TYPE ST_TCUEPT :
STRUCT
	// LoadPort module state 
	//arrLPSubModule : ARRAY [1..(.NO_OF_LANES)] OF ST_LP_SubModuleEPT;
	// Vision Shuttle 
	TCU : E_EPT;
END_STRUCT
END_TYPE

(* stored: Version 1.1.0.1, ProductVersion 3.1.4022.12
   DUT ST_TCUEPT: Id {9f00026a-a904-41aa-bc64-905de90e5a87} *)
